TYPE MAIN_BUSY :
(
	eMainWaitStart := 0
);
END_TYPE

(* stored: Version 1.1.0.1, ProductVersion 3.1.4024.2
   DUT MAIN_BUSY: Id {c3b478f4-370b-4219-a0df-85b8f47a8821} *)
